(* Schneider Machine Expert - Basic project 友成插座（５个点）检测带２个安全门加开关检测 , file version 1.6.0.0 *)
(* ProjectInformations: Name=New project *)

HARDWARE
  Cpu 0: TM221CE40T
  EthernetConfiguration: NetworkName=M221, IpAllocationMode=FixedAddress, IpAddress=0.0.0.0, SubnetMask=0.0.0.0
  SerialLineConfiguration: Baud=Baud19200, Parity=ParityEven, DataBits=DataBits8, StopBits=StopBits1, PhysicalMedium=PhysicalMediumRs485, TransmissionMode=TransmissionModeModbusRtu, SlaveId=1, Addressing=SlaveAddressing
  MastTask: UsePeriodScanMode=false, PeriodScan=100
  FastTask: Period=255
  CpuBehavior: StartingMode=StartAsPreviousState, AutoSaveRamOnEeprom=true, WatchdogPeriod=250

SYMBOLS  (address, symbol, comment, settings)
  %M0         "左按钮"
  %M1         "右按钮"
  %M2         "拉料进到位感应"
  %M3         "伺服上限"
  %M4         "伺服中间感应位"
  %M5         "伺服下限"
  %M6         "机器安全门开关"
  %M7         "面板复位按扭"
  %M8         "面板停止按扭"
  %M9         "拉P汽缸到位"
  %M10        "導通1"
  %M11        "導通2"
  %M12        "導通3"
  %M13        "導通4"
  %M14        "導通5"
  %M16        "安全门检测1"
  %M17        "安全门检测2"
  %M50        "运行开始"
  %M51        "导通OK"
  %M52        "导通NG"
  %M53        "产品OK"
  %M54        "产品NG"
  %M55        "拉P汽缸輔助"
  %M56        "开关 关OK"
  %M57        "开关 关NG"
  %M58        "开关 开OK"
  %M59        "开关 开NG"
  %M104       "双手启动按扭指示灯"
  %M105       "报警指示灯"
  %M106       "OK指示灯"
  %M107       "NG指示灯"
  %M108       "蜂鸣器"
  %M109       "拉料进汽缸"
  %M110       "拉P汽缸"
  %M111       "拉P汽缸延時輔助"
  %M112       "开关 开"
  %M113       "开关 关"
  %M209       "电机向下"
  %M210       "电机向方向"
  %M213       "電機向上"
  %M215       "電機向下輔助"
  %S0       SB_COLDSTART  "Indicates or executes a cold start (data initialized to default values)"
  %S1       SB_WARMSTART  "Indicates there was a warm start with data backup"
  %S6       SB_TB1S  "Time base of 1 s generated by an internal clock"
  %S13      SB_FIRSTRUN  "Indicates the first controller cycle in RUN mode"
  %TM0        [Preset=5, Base=OneHundredMilliSeconds]
  %TM1        [Preset=5, Base=OneHundredMilliSeconds]
  %TM3        [Preset=8, Base=OneHundredMilliSeconds]
  %TM4        [Preset=5, Base=OneHundredMilliSeconds]
  %TM5        [Preset=5, Base=OneHundredMilliSeconds]
  %TM6        [Preset=5, Base=OneHundredMilliSeconds]
  %TM7        [Preset=5, Base=OneHundredMilliSeconds]
  %TM8        [Preset=10, Base=OneHundredMilliSeconds]
  %TM9        [Preset=5, Base=OneHundredMilliSeconds]
  %TM10       [Preset=10, Base=OneHundredMilliSeconds]
  %I0.0       "左按钮"
  %I0.1       "右按钮"
  %I0.2       "拉料进到位感应"
  %I0.3       "伺服上限"
  %I0.4       "伺服下限"
  %I0.5       "伺服下限"
  %I0.6       "机器安全门开关"
  %I0.7       "面板复位按扭"
  %I0.8       "面板停止按扭"
  %I0.9       "拉P汽缸到位"
  %I0.16      "安全门检测1"
  %I0.17      "安全门检测2"
  %Q0.1       "脉冲方向"
  %Q0.4       "双手启动按扭指示灯"
  %Q0.5       "报警指示灯"
  %Q0.6       "OK指示灯"
  %Q0.7       "NG指示灯"
  %Q0.8       "蜂鸣器"
  %Q0.9       "拉料进汽缸"
  %Q0.10      "拉P汽缸"
  %Q0.11      "下顶"
  %PLS0       [PtoObject(RefInput=NotUsed, ZPhaseInput=NotUsed, ProbeInput=NotUsed), GlobalIndex=0, Type=PLS, TimeBase=ZeroPointOneMilliSeconds, Preset=1, UseDoubleWord=true]

POU 新 POU
  (* SectionNumber=1 *)

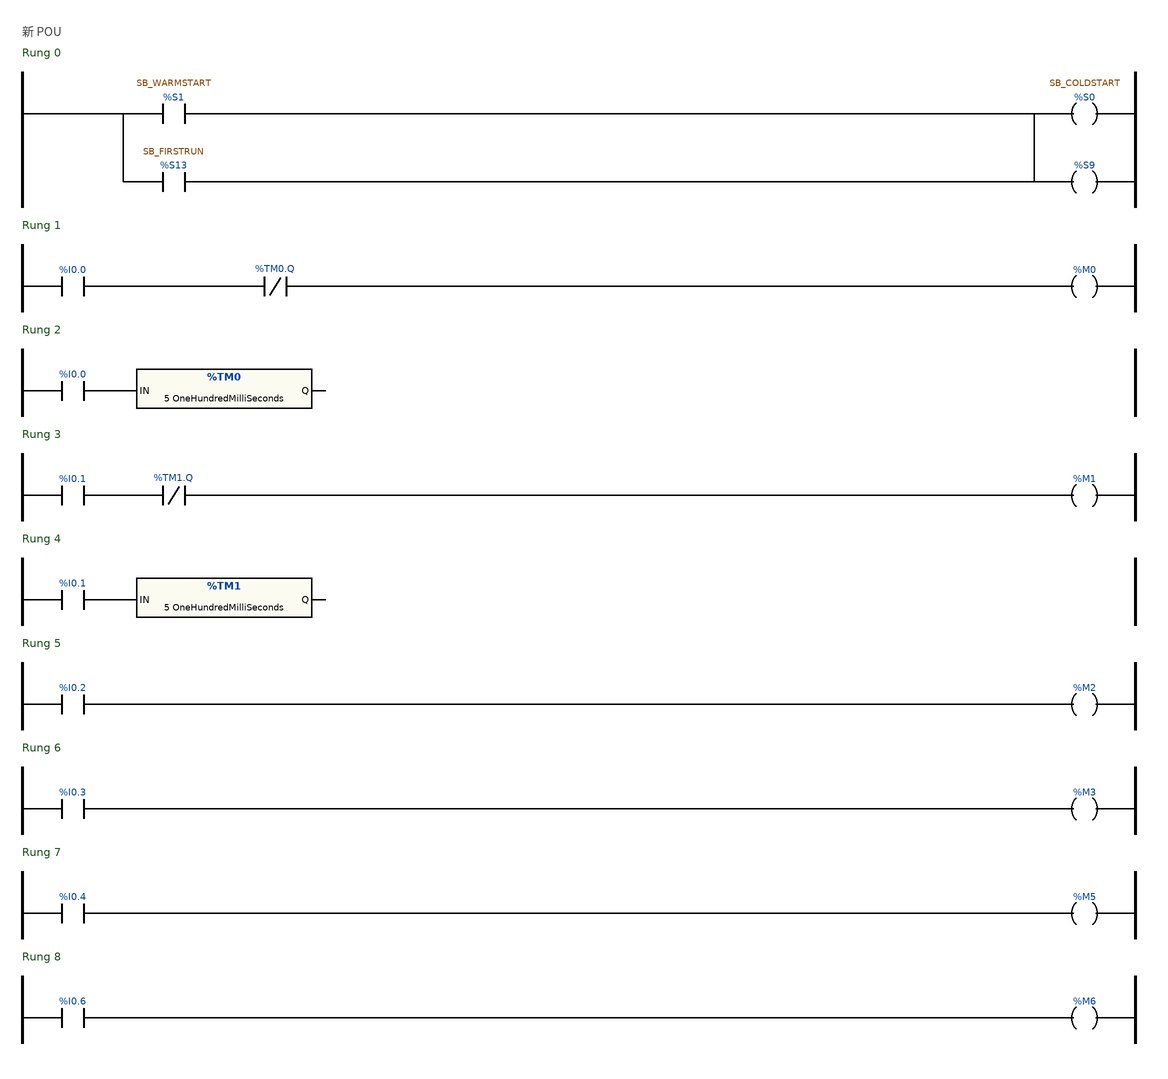

// Rung 0
  LD %S1                  (* SB_WARMSTART *)
  OR %S13                 (* SB_FIRSTRUN *)
  ST %S0                  (* SB_COLDSTART *)
  ST %S9
  // as ST:
  //   SB_COLDSTART := SB_WARMSTART OR SB_FIRSTRUN;
  //   %S9 := SB_WARMSTART OR SB_FIRSTRUN;

// Rung 1
  LD %I0.0
  ANDN %TM0.Q
  ST %M0
  // as ST:
  //   %M0 := %I0.0 AND NOT %TM0.Q;

// Rung 2
  BLK %TM0
  LD %I0.0
  IN
  END_BLK
  // as ST:
  //   %TM0(IN := %I0.0);

// Rung 3
  LD %I0.1
  ANDN %TM1.Q
  ST %M1
  // as ST:
  //   %M1 := %I0.1 AND NOT %TM1.Q;

// Rung 4
  BLK %TM1
  LD %I0.1
  IN
  END_BLK
  // as ST:
  //   %TM1(IN := %I0.1);

// Rung 5
  LD %I0.2
  ST %M2
  // as ST:
  //   %M2 := %I0.2;

// Rung 6
  LD %I0.3
  ST %M3
  // as ST:
  //   %M3 := %I0.3;

// Rung 7
  LD %I0.4
  ST %M5
  // as ST:
  //   %M5 := %I0.4;

// Rung 8
  LD %I0.6
  ST %M6
  // as ST:
  //   %M6 := %I0.6;

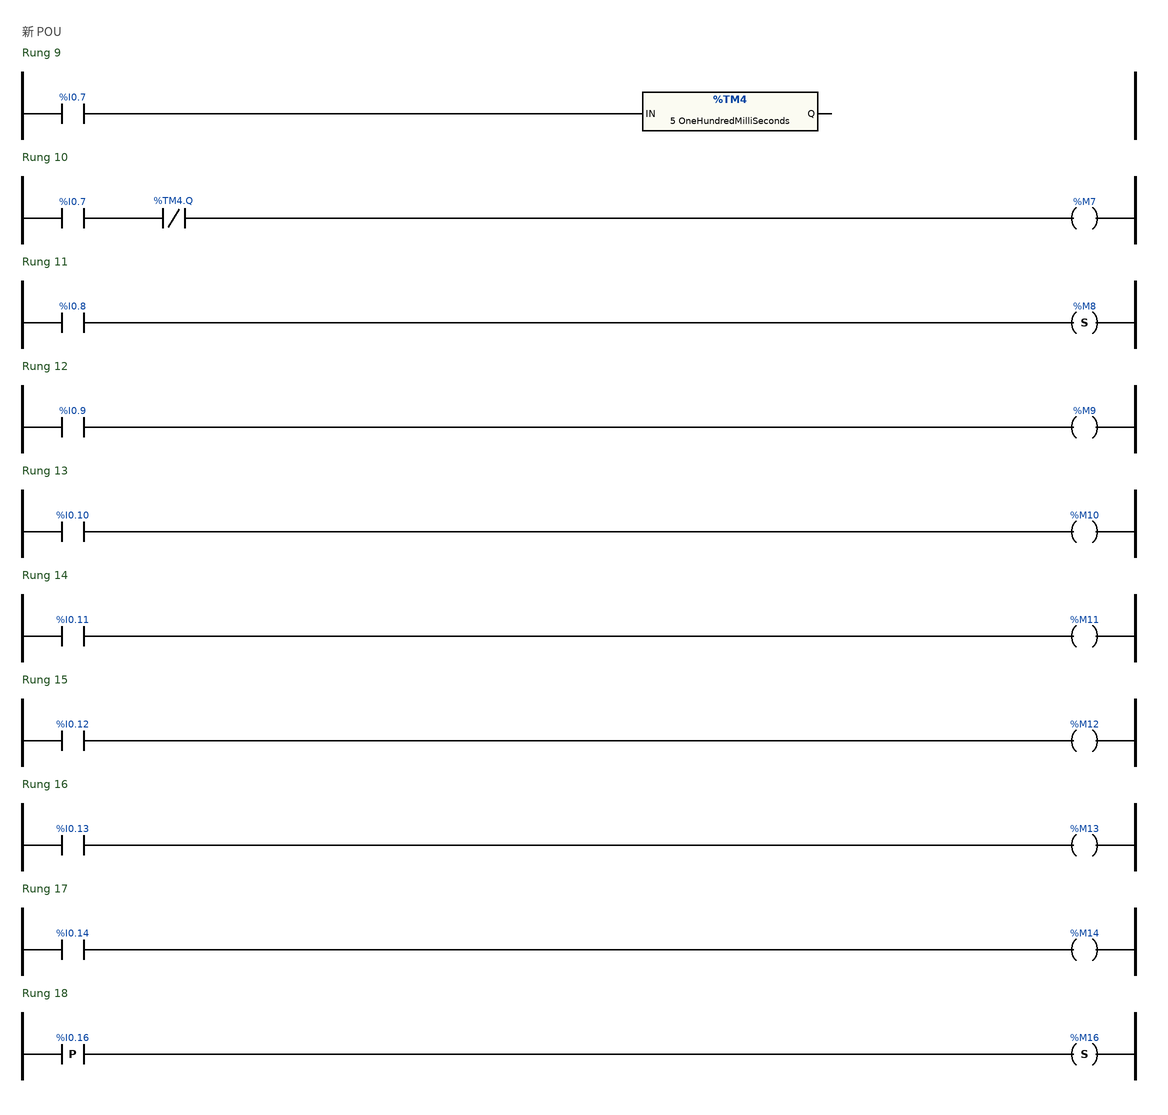

// Rung 9
  BLK %TM4
  LD %I0.7
  IN
  END_BLK
  // as ST:
  //   %TM4(IN := %I0.7);

// Rung 10
  LD %I0.7
  ANDN %TM4.Q
  ST %M7
  // as ST:
  //   %M7 := %I0.7 AND NOT %TM4.Q;

// Rung 11
  LD %I0.8
  S %M8
  // as ST:
  //   IF %I0.8 THEN %M8 := TRUE; END_IF;

// Rung 12
  LD %I0.9
  ST %M9
  // as ST:
  //   %M9 := %I0.9;

// Rung 13
  LD %I0.10
  ST %M10
  // as ST:
  //   %M10 := %I0.10;

// Rung 14
  LD %I0.11
  ST %M11
  // as ST:
  //   %M11 := %I0.11;

// Rung 15
  LD %I0.12
  ST %M12
  // as ST:
  //   %M12 := %I0.12;

// Rung 16
  LD %I0.13
  ST %M13
  // as ST:
  //   %M13 := %I0.13;

// Rung 17
  LD %I0.14
  ST %M14
  // as ST:
  //   %M14 := %I0.14;

// Rung 18
  LDR %I0.16
  S %M16
  // as ST:
  //   IF RISING(%I0.16) THEN %M16 := TRUE; END_IF;

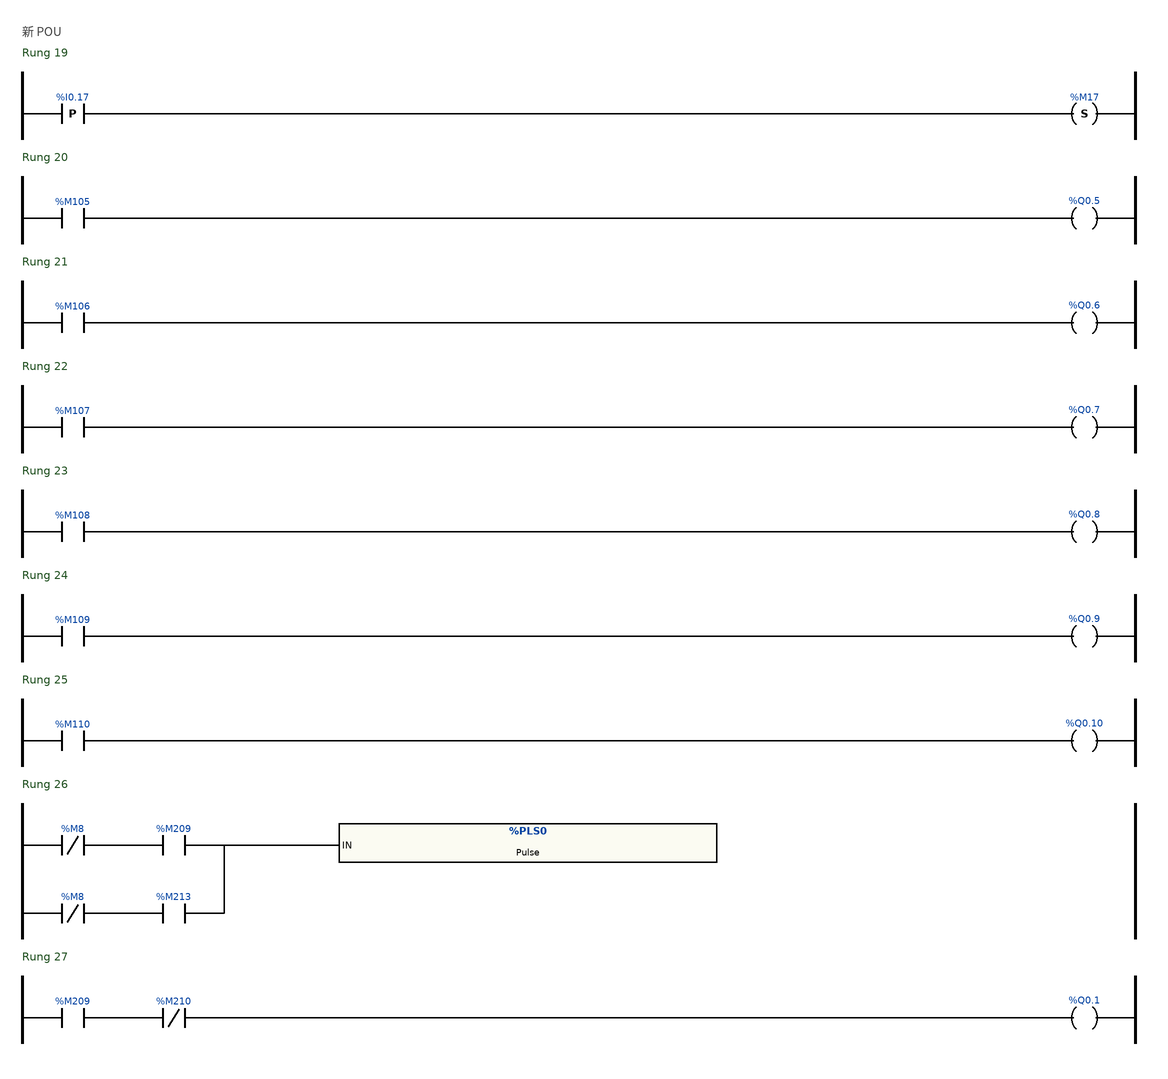

// Rung 19
  LDR %I0.17
  S %M17
  // as ST:
  //   IF RISING(%I0.17) THEN %M17 := TRUE; END_IF;

// Rung 20
  LD %M105
  ST %Q0.5
  // as ST:
  //   %Q0.5 := %M105;

// Rung 21
  LD %M106
  ST %Q0.6
  // as ST:
  //   %Q0.6 := %M106;

// Rung 22
  LD %M107
  ST %Q0.7
  // as ST:
  //   %Q0.7 := %M107;

// Rung 23
  LD %M108
  ST %Q0.8
  // as ST:
  //   %Q0.8 := %M108;

// Rung 24
  LD %M109
  ST %Q0.9
  // as ST:
  //   %Q0.9 := %M109;

// Rung 25
  LD %M110
  ST %Q0.10
  // as ST:
  //   %Q0.10 := %M110;

// Rung 26
  BLK %PLS0
  LDN %M8
  AND %M209
  OR(N %M8
  AND %M213
  )
  IN
  END_BLK
  // as ST:
  //   %PLS0(IN := NOT %M8 AND %M209 OR NOT %M8 AND %M213);

// Rung 27
  LD %M209
  ANDN %M210
  ST %Q0.1
  // as ST:
  //   %Q0.1 := %M209 AND NOT %M210;

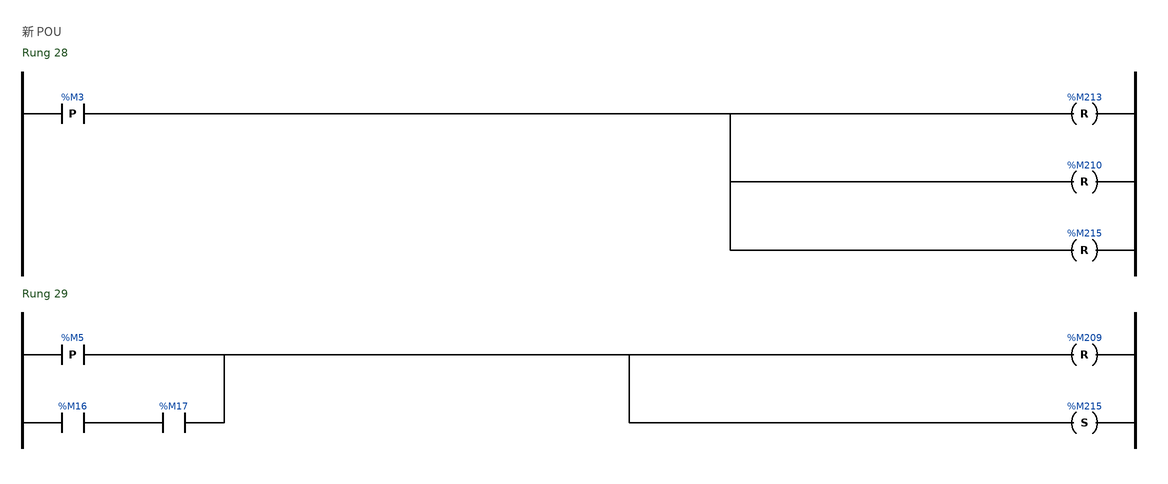

// Rung 28
  LDR %M3
  R %M213
  R %M210
  R %M215
  // as ST:
  //   IF RISING(%M3) THEN %M213 := FALSE; END_IF;
  //   IF RISING(%M3) THEN %M210 := FALSE; END_IF;
  //   IF RISING(%M3) THEN %M215 := FALSE; END_IF;

// Rung 29
  LDR %M5
  OR( %M16
  AND %M17
  )
  R %M209
  S %M215
  // as ST:
  //   IF RISING(%M5) OR %M16 AND %M17 THEN %M209 := FALSE; END_IF;
  //   IF RISING(%M5) OR %M16 AND %M17 THEN %M215 := TRUE; END_IF;

POU 新 POU
  (* SectionNumber=2 *)

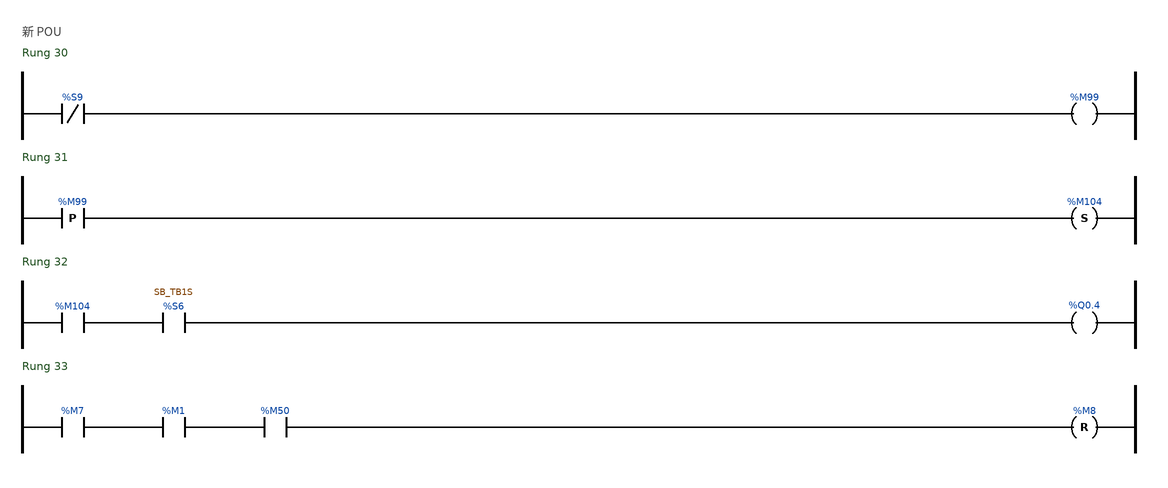

// Rung 30
  LDN %S9
  ST %M99
  // as ST:
  //   %M99 := NOT %S9;

// Rung 31
  LDR %M99
  S %M104
  // as ST:
  //   IF RISING(%M99) THEN %M104 := TRUE; END_IF;

// Rung 32
  LD %M104
  AND %S6                 (* SB_TB1S *)
  ST %Q0.4
  // as ST:
  //   %Q0.4 := %M104 AND SB_TB1S;

// Rung 33
  LD %M7
  AND %M1
  AND %M50
  R %M8
  // as ST:
  //   IF %M7 AND %M1 AND %M50 THEN %M8 := FALSE; END_IF;

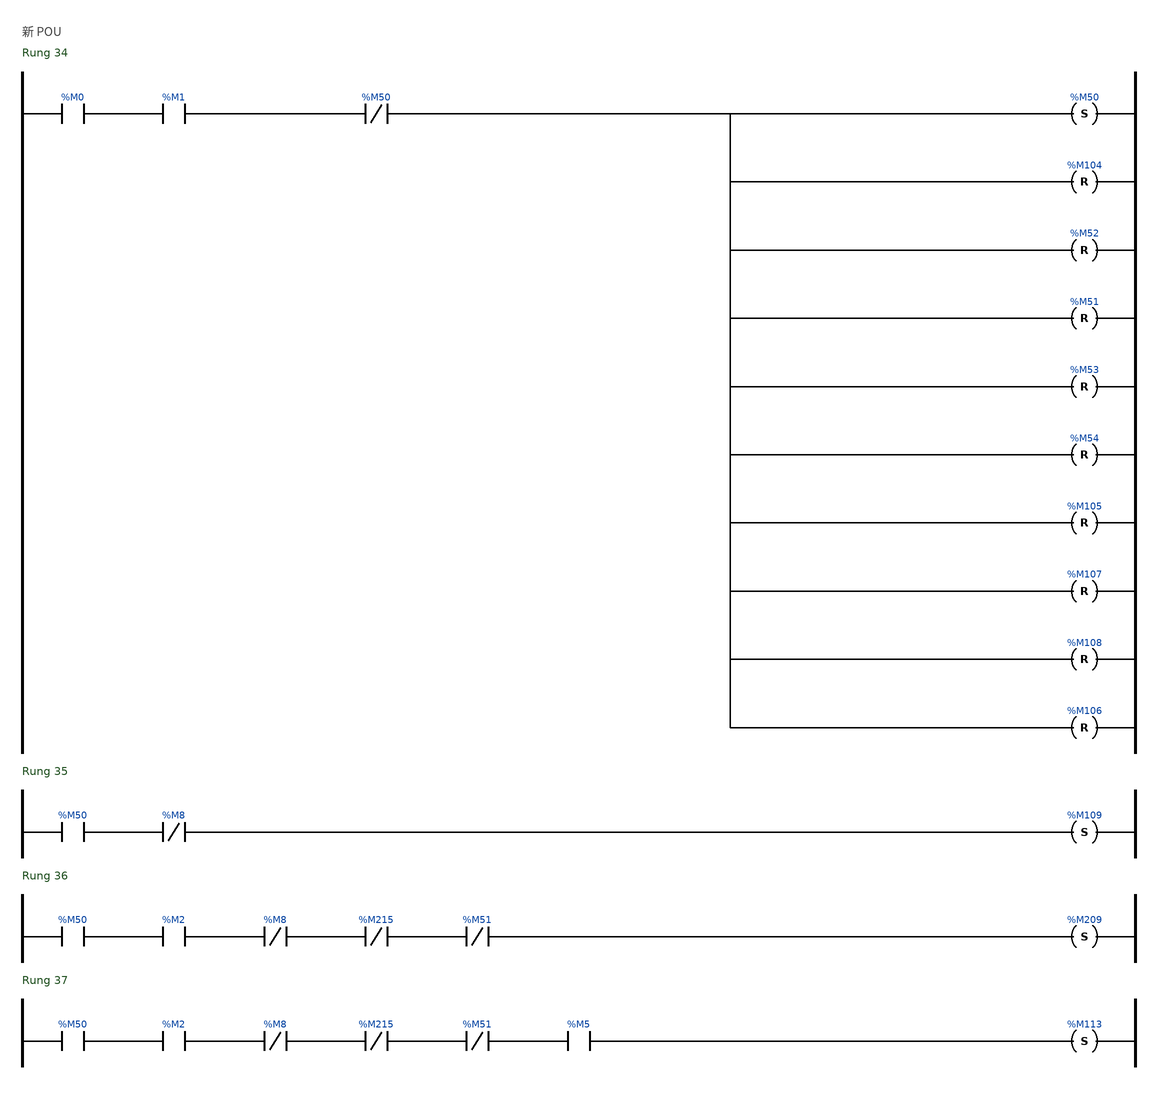

// Rung 34
  LD %M0
  AND %M1
  ANDN %M50
  S %M50
  R %M104
  R %M52
  R %M51
  R %M53
  R %M54
  R %M105
  R %M107
  R %M108
  R %M106
  // as ST:
  //   _t1 := %M0 AND %M1 AND NOT %M50;
  //   IF _t1 THEN %M50 := TRUE; END_IF;
  //   IF _t1 THEN %M104 := FALSE; END_IF;
  //   IF _t1 THEN %M52 := FALSE; END_IF;
  //   IF _t1 THEN %M51 := FALSE; END_IF;
  //   IF _t1 THEN %M53 := FALSE; END_IF;
  //   IF _t1 THEN %M54 := FALSE; END_IF;
  //   IF _t1 THEN %M105 := FALSE; END_IF;
  //   IF _t1 THEN %M107 := FALSE; END_IF;
  //   IF _t1 THEN %M108 := FALSE; END_IF;
  //   IF _t1 THEN %M106 := FALSE; END_IF;

// Rung 35
  LD %M50
  ANDN %M8
  S %M109
  // as ST:
  //   IF %M50 AND NOT %M8 THEN %M109 := TRUE; END_IF;

// Rung 36
  LD %M50
  AND %M2
  ANDN %M8
  ANDN %M215
  ANDN %M51
  S %M209
  // as ST:
  //   IF %M50 AND %M2 AND NOT %M8 AND NOT %M215 AND NOT %M51 THEN %M209 := TRUE; END_IF;

// Rung 37
  LD %M50
  AND %M2
  ANDN %M8
  ANDN %M215
  ANDN %M51
  AND %M5
  S %M113
  // as ST:
  //   IF %M50 AND %M2 AND NOT %M8 AND NOT %M215 AND NOT %M51 AND %M5 THEN %M113 := TRUE; END_IF;

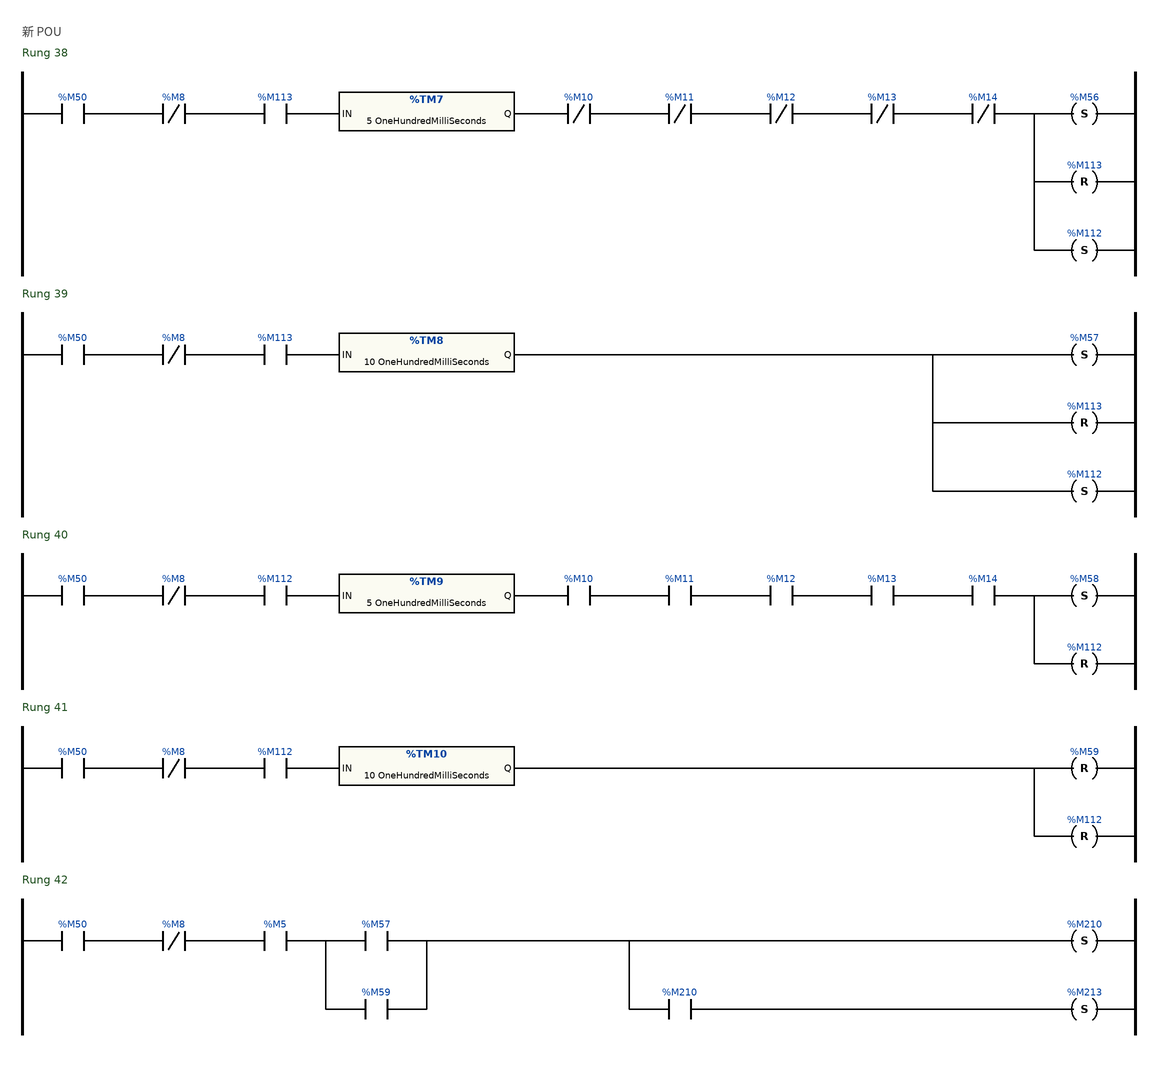

// Rung 38
  BLK %TM7
  LD %M50
  ANDN %M8
  AND %M113
  IN
  OUT_BLK
  LD Q
  ANDN %M10
  ANDN %M11
  ANDN %M12
  ANDN %M13
  ANDN %M14
  S %M56
  R %M113
  S %M112
  END_BLK
  // as ST:
  //   %TM7(IN := %M50 AND NOT %M8 AND %M113);
  //   IF %TM7.Q AND NOT %M10 AND NOT %M11 AND NOT %M12 AND NOT %M13 AND NOT %M14 THEN %M56 := TRUE; END_IF;
  //   IF %TM7.Q AND NOT %M10 AND NOT %M11 AND NOT %M12 AND NOT %M13 AND NOT %M14 THEN %M113 := FALSE; END_IF;
  //   IF %TM7.Q AND NOT %M10 AND NOT %M11 AND NOT %M12 AND NOT %M13 AND NOT %M14 THEN %M112 := TRUE; END_IF;

// Rung 39
  BLK %TM8
  LD %M50
  ANDN %M8
  AND %M113
  IN
  OUT_BLK
  LD Q
  S %M57
  R %M113
  S %M112
  END_BLK
  // as ST:
  //   %TM8(IN := %M50 AND NOT %M8 AND %M113);
  //   IF %TM8.Q THEN %M57 := TRUE; END_IF;
  //   IF %TM8.Q THEN %M113 := FALSE; END_IF;
  //   IF %TM8.Q THEN %M112 := TRUE; END_IF;

// Rung 40
  BLK %TM9
  LD %M50
  ANDN %M8
  AND %M112
  IN
  OUT_BLK
  LD Q
  AND %M10
  AND %M11
  AND %M12
  AND %M13
  AND %M14
  S %M58
  R %M112
  END_BLK
  // as ST:
  //   %TM9(IN := %M50 AND NOT %M8 AND %M112);
  //   IF %TM9.Q AND %M10 AND %M11 AND %M12 AND %M13 AND %M14 THEN %M58 := TRUE; END_IF;
  //   IF %TM9.Q AND %M10 AND %M11 AND %M12 AND %M13 AND %M14 THEN %M112 := FALSE; END_IF;

// Rung 41
  BLK %TM10
  LD %M50
  ANDN %M8
  AND %M112
  IN
  OUT_BLK
  LD Q
  R %M59
  R %M112
  END_BLK
  // as ST:
  //   %TM10(IN := %M50 AND NOT %M8 AND %M112);
  //   IF %TM10.Q THEN %M59 := FALSE; END_IF;
  //   IF %TM10.Q THEN %M112 := FALSE; END_IF;

// Rung 42
  LD %M50
  ANDN %M8
  AND %M5
  AND( %M57
  OR %M59
  )
  MPS
  S %M210
  MPP
  AND %M210
  S %M213
  // as ST:
  //   IF %M50 AND NOT %M8 AND %M5 AND (%M57 OR %M59) THEN %M210 := TRUE; END_IF;
  //   IF %M50 AND NOT %M8 AND %M5 AND (%M57 OR %M59) AND %M210 THEN %M213 := TRUE; END_IF;

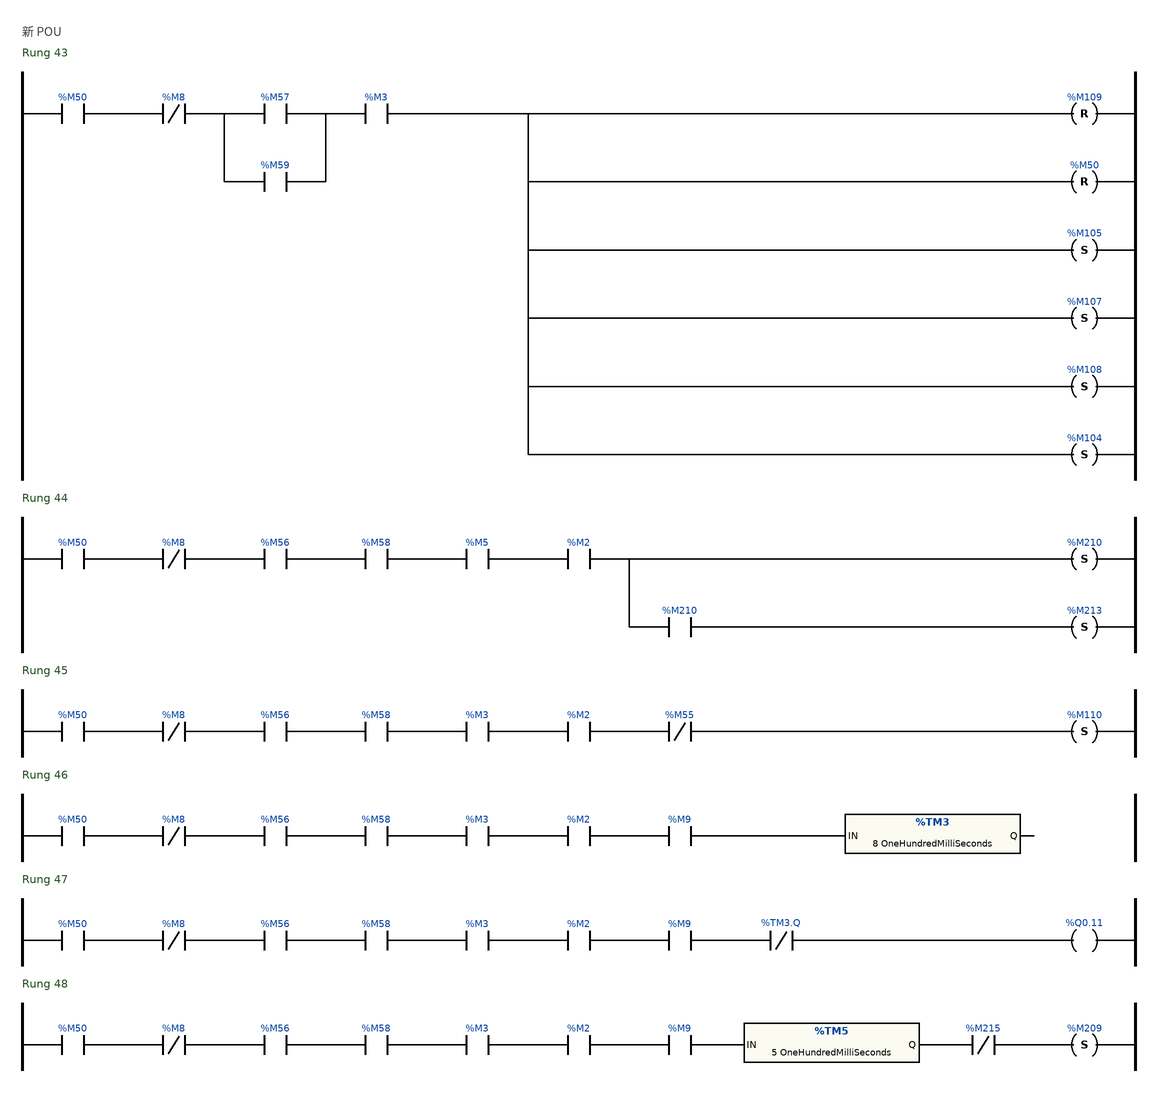

// Rung 43
  LD %M50
  ANDN %M8
  AND( %M57
  OR %M59
  )
  AND %M3
  R %M109
  R %M50
  S %M105
  S %M107
  S %M108
  S %M104
  // as ST:
  //   IF %M50 AND NOT %M8 AND (%M57 OR %M59) AND %M3 THEN %M109 := FALSE; END_IF;
  //   _t1 := %M50 AND NOT %M8 AND (%M57 OR %M59) AND %M3;
  //   IF _t1 THEN %M50 := FALSE; END_IF;
  //   IF _t1 THEN %M105 := TRUE; END_IF;
  //   IF _t1 THEN %M107 := TRUE; END_IF;
  //   IF _t1 THEN %M108 := TRUE; END_IF;
  //   IF _t1 THEN %M104 := TRUE; END_IF;

// Rung 44
  LD %M50
  ANDN %M8
  AND %M56
  AND %M58
  AND %M5
  AND %M2
  MPS
  S %M210
  MPP
  AND %M210
  S %M213
  // as ST:
  //   IF %M50 AND NOT %M8 AND %M56 AND %M58 AND %M5 AND %M2 THEN %M210 := TRUE; END_IF;
  //   IF %M50 AND NOT %M8 AND %M56 AND %M58 AND %M5 AND %M2 AND %M210 THEN %M213 := TRUE; END_IF;

// Rung 45
  LD %M50
  ANDN %M8
  AND %M56
  AND %M58
  AND %M3
  AND %M2
  ANDN %M55
  S %M110
  // as ST:
  //   IF %M50 AND NOT %M8 AND %M56 AND %M58 AND %M3 AND %M2 AND NOT %M55 THEN %M110 := TRUE; END_IF;

// Rung 46
  BLK %TM3
  LD %M50
  ANDN %M8
  AND %M56
  AND %M58
  AND %M3
  AND %M2
  AND %M9
  IN
  END_BLK
  // as ST:
  //   %TM3(IN := %M50 AND NOT %M8 AND %M56 AND %M58 AND %M3 AND %M2 AND %M9);

// Rung 47
  LD %M50
  ANDN %M8
  AND %M56
  AND %M58
  AND %M3
  AND %M2
  AND %M9
  ANDN %TM3.Q
  ST %Q0.11
  // as ST:
  //   %Q0.11 := %M50 AND NOT %M8 AND %M56 AND %M58 AND %M3 AND %M2 AND %M9 AND NOT %TM3.Q;

// Rung 48
  BLK %TM5
  LD %M50
  ANDN %M8
  AND %M56
  AND %M58
  AND %M3
  AND %M2
  AND %M9
  IN
  OUT_BLK
  LD Q
  ANDN %M215
  S %M209
  END_BLK
  // as ST:
  //   %TM5(IN := %M50 AND NOT %M8 AND %M56 AND %M58 AND %M3 AND %M2 AND %M9);
  //   IF %TM5.Q AND NOT %M215 THEN %M209 := TRUE; END_IF;

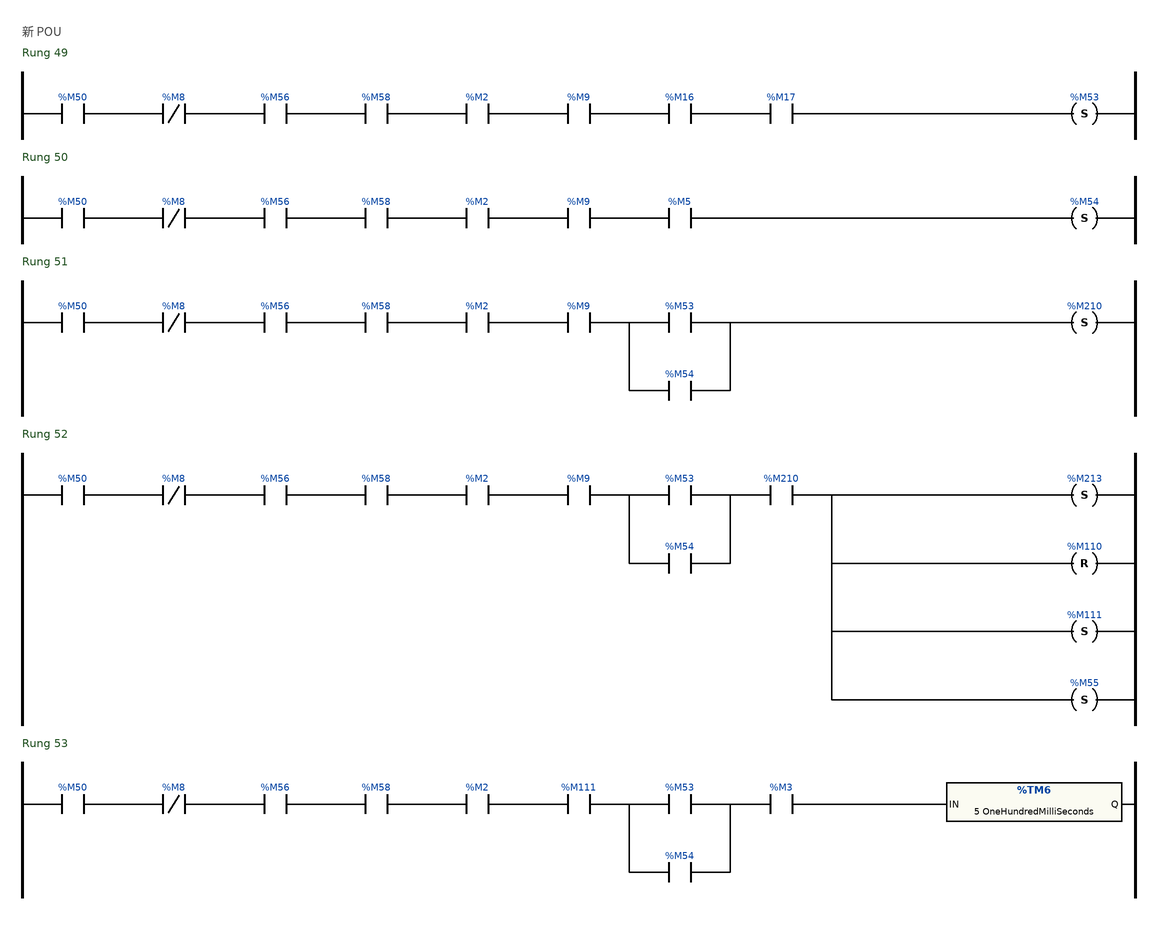

// Rung 49
  LD %M50
  ANDN %M8
  AND %M56
  AND %M58
  AND %M2
  AND %M9
  AND %M16
  AND %M17
  S %M53
  // as ST:
  //   IF %M50 AND NOT %M8 AND %M56 AND %M58 AND %M2 AND %M9 AND %M16 AND %M17 THEN %M53 := TRUE; END_IF;

// Rung 50
  LD %M50
  ANDN %M8
  AND %M56
  AND %M58
  AND %M2
  AND %M9
  AND %M5
  S %M54
  // as ST:
  //   IF %M50 AND NOT %M8 AND %M56 AND %M58 AND %M2 AND %M9 AND %M5 THEN %M54 := TRUE; END_IF;

// Rung 51
  LD %M50
  ANDN %M8
  AND %M56
  AND %M58
  AND %M2
  AND %M9
  AND( %M53
  OR %M54
  )
  S %M210
  // as ST:
  //   IF %M50 AND NOT %M8 AND %M56 AND %M58 AND %M2 AND %M9 AND (%M53 OR %M54) THEN %M210 := TRUE; END_IF;

// Rung 52
  LD %M50
  ANDN %M8
  AND %M56
  AND %M58
  AND %M2
  AND %M9
  AND( %M53
  OR %M54
  )
  AND %M210
  S %M213
  R %M110
  S %M111
  S %M55
  // as ST:
  //   IF %M50 AND NOT %M8 AND %M56 AND %M58 AND %M2 AND %M9 AND (%M53 OR %M54) AND %M210 THEN %M213 := TRUE; END_IF;
  //   IF %M50 AND NOT %M8 AND %M56 AND %M58 AND %M2 AND %M9 AND (%M53 OR %M54) AND %M210 THEN %M110 := FALSE; END_IF;
  //   IF %M50 AND NOT %M8 AND %M56 AND %M58 AND %M2 AND %M9 AND (%M53 OR %M54) AND %M210 THEN %M111 := TRUE; END_IF;
  //   IF %M50 AND NOT %M8 AND %M56 AND %M58 AND %M2 AND %M9 AND (%M53 OR %M54) AND %M210 THEN %M55 := TRUE; END_IF;

// Rung 53
  BLK %TM6
  LD %M50
  ANDN %M8
  AND %M56
  AND %M58
  AND %M2
  AND %M111
  AND( %M53
  OR %M54
  )
  AND %M3
  IN
  END_BLK
  // as ST:
  //   %TM6(IN := %M50 AND NOT %M8 AND %M56 AND %M58 AND %M2 AND %M111 AND (%M53 OR %M54) AND %M3);

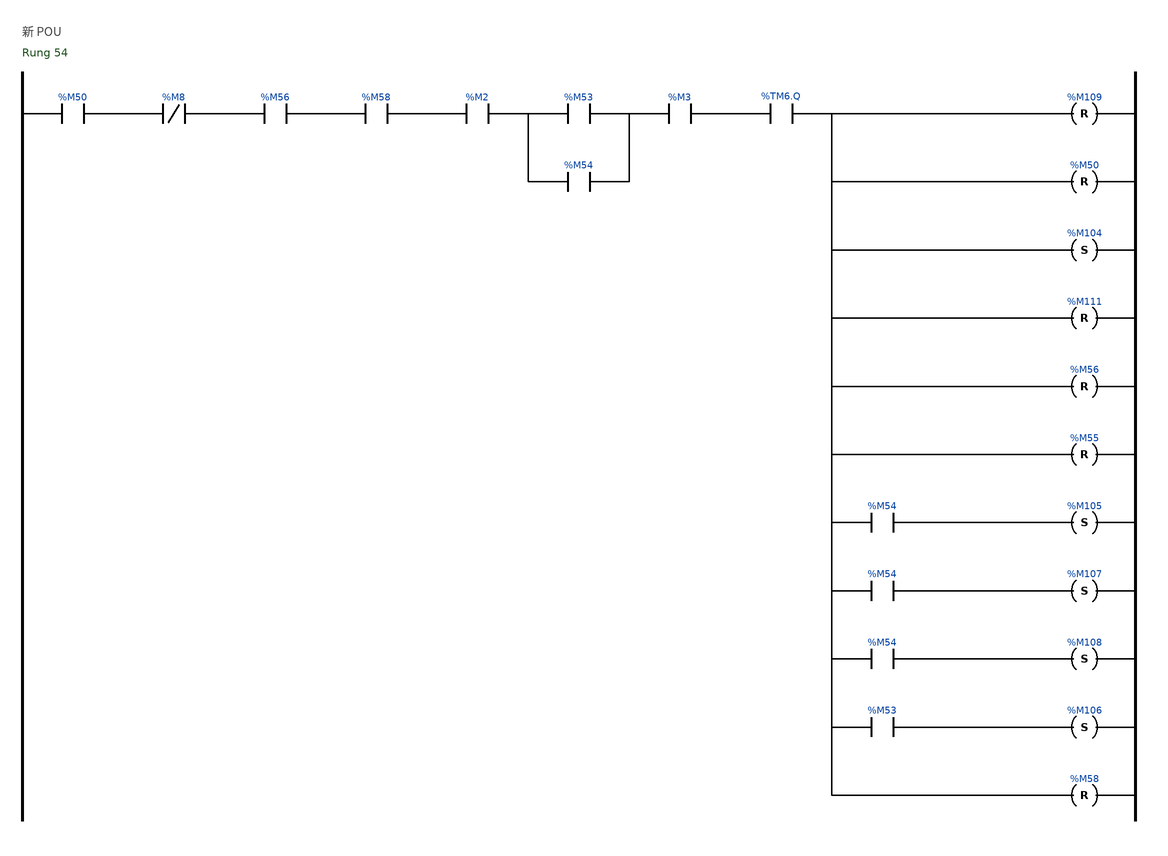

// Rung 54
  LD %M50
  ANDN %M8
  AND %M56
  AND %M58
  AND %M2
  AND( %M53
  OR %M54
  )
  AND %M3
  AND %TM6.Q
  MPS
  R %M109
  MRD
  R %M50
  MRD
  S %M104
  MRD
  R %M111
  MRD
  R %M56
  MRD
  R %M55
  MRD
  AND %M54
  S %M105
  MRD
  AND %M54
  S %M107
  MRD
  AND %M54
  S %M108
  MRD
  AND %M53
  S %M106
  MPP
  R %M58
  // as ST:
  //   IF %M50 AND NOT %M8 AND %M56 AND %M58 AND %M2 AND (%M53 OR %M54) AND %M3 AND %TM6.Q THEN %M109 := FALSE; END_IF;
  //   _t1 := %M50 AND NOT %M8 AND %M56 AND %M58 AND %M2 AND (%M53 OR %M54) AND %M3 AND %TM6.Q;
  //   IF _t1 THEN %M50 := FALSE; END_IF;
  //   IF _t1 THEN %M104 := TRUE; END_IF;
  //   IF _t1 THEN %M111 := FALSE; END_IF;
  //   IF _t1 THEN %M56 := FALSE; END_IF;
  //   IF _t1 THEN %M55 := FALSE; END_IF;
  //   IF _t1 AND %M54 THEN %M105 := TRUE; END_IF;
  //   IF _t1 AND %M54 THEN %M107 := TRUE; END_IF;
  //   IF _t1 AND %M54 THEN %M108 := TRUE; END_IF;
  //   IF _t1 AND %M53 THEN %M106 := TRUE; END_IF;
  //   IF _t1 THEN %M58 := FALSE; END_IF;
